// TIA Portal project "FanGas_Combustion" (V17)

(* hardware
DEVICE "PLC_1"  S7-1200 Station
   slot 0: "Rack_0"  S7-1200 Rack  Rack  V1.0
   slot 1: "PLC_1"  CPU 1214C AC/DC/Rly  6ES7 214-1BG40-0XB0  V4.5
*)

// ===== PLC "PLC_1"  CPU 1214C AC/DC/Rly =====

VAR_GLOBAL   // PLC tag table "PLC_tags"
   "风机运行" AT %Q4.4 : Bool;
   "烧嘴电源" AT %Q4.6 : Bool;
   "风机控制" AT %QW44 : Int;
END_VAR

DATA_BLOCK "信号数据"   // DB1
{ S7_Optimized_Access := 'TRUE' }
VERSION : 0.1
   VAR
      风机运行按 : Bool;   // 风机运行按钮
      风机故障反馈 : Bool;   // 风机故障反馈信号
      风机手动 : Bool;   // 风机手动模式选择
      风机自动输出 : Real;   // 风机自动控制输出值
      风机手动频率 : Real;   // 风机手动频率设定
      风机控制输出 : Real;   // 风机最终控制输出
      风压测量值 : Real;   // 风压传感器测量值
   END_VAR
BEGIN
END_DATA_BLOCK

DATA_BLOCK "内部数据"   // DB2
{ S7_Optimized_Access := 'TRUE' }
VERSION : 0.1
   VAR
      风机控制输出值 : Real;   // 风机频率百分比对应的0-27648中间值
      风压过渡 : Int;   // 风压模拟量输出过渡值
   END_VAR
BEGIN
END_DATA_BLOCK

FUNCTION "FC_FanGasControl" : Void   // FC1, LAD
{ S7_Optimized_Access := 'TRUE' }
BEGIN

REGION Network 1: 风机输出
   // 风机运行按常开+风机故障反馈常闭→风机运行线圈；手动选择MOVE自动输出或MUL手动频率×2→控制输出
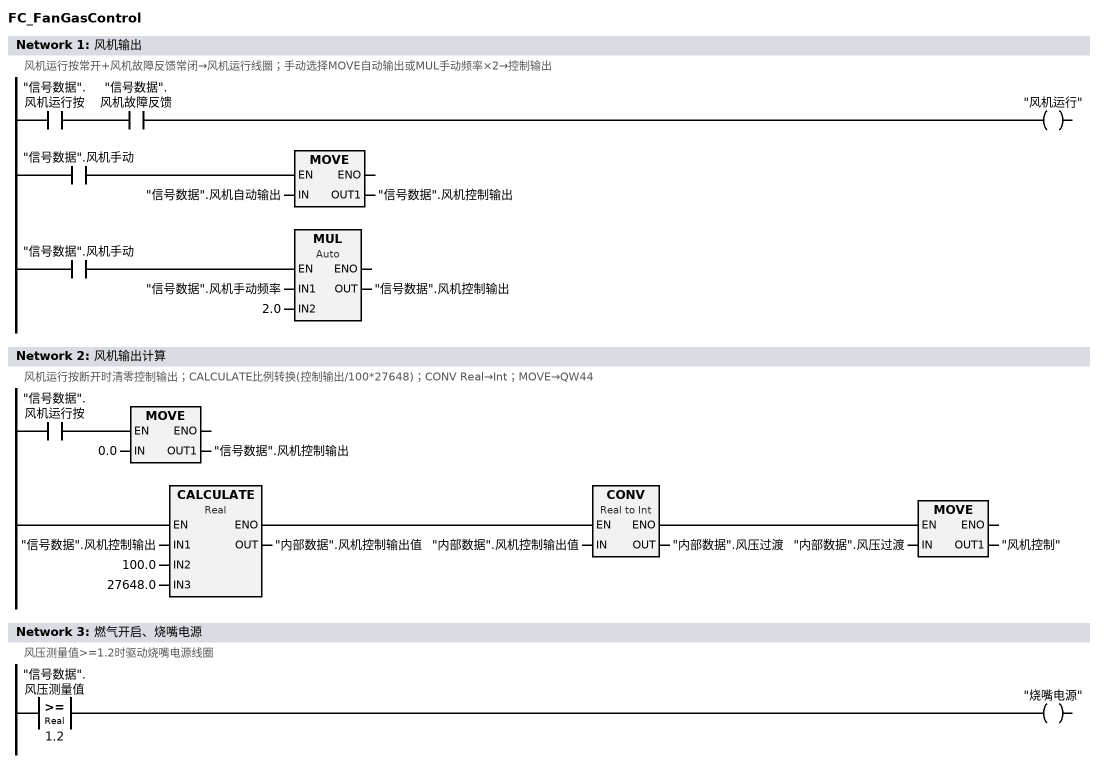
   RUNG wire#powerrail
      Contact( "信号数据".风机运行按 )
      Contact( "信号数据".风机故障反馈 )
      Coil( "风机运行" )
   END_RUNG
   RUNG wire#powerrail
      Contact( "信号数据".风机手动 )
      Move(in := "信号数据".风机自动输出, out1 => "信号数据".风机控制输出)
   END_RUNG
   RUNG wire#powerrail
      Contact( "信号数据".风机手动 )
      Mul(in1 := "信号数据".风机手动频率, in2 := 2.0, out => "信号数据".风机控制输出)
   END_RUNG
   // the same network as SCL:
   "风机运行" := "信号数据".风机运行按 AND "信号数据".风机故障反馈;
   IF "信号数据".风机手动 THEN
       "信号数据".风机控制输出 := "信号数据".风机自动输出;
       "信号数据".风机控制输出 := "信号数据".风机手动频率 * 2.0;
   END_IF;
END_REGION

REGION Network 2: 风机输出计算
   // 风机运行按断开时清零控制输出；CALCULATE比例转换(控制输出/100*27648)；CONV Real→Int；MOVE→QW44
   RUNG wire#powerrail
      Contact( "信号数据".风机运行按 )
      Move(in := 0.0, out1 => "信号数据".风机控制输出)
   END_RUNG
   RUNG wire#powerrail
      { S7_Templates := "SrcType := Real"; S7_Expression := "(IN1/IN2)*IN3" } Calculate(in1 := "信号数据".风机控制输出, in2 := 100.0, in3 := 27648.0, out => "内部数据".风机控制输出值)
      { S7_Templates := "[SrcType := Real, DestType := Int]" } Convert(in := "内部数据".风机控制输出值, out => "内部数据".风压过渡)
      Move(in := "内部数据".风压过渡, out1 => "风机控制")
   END_RUNG
   // the same network as SCL:
   IF "信号数据".风机运行按 THEN "信号数据".风机控制输出 := 0.0; END_IF;
   "内部数据".风机控制输出值 := ("信号数据".风机控制输出/100.0)*27648.0;
   "内部数据".风压过渡 := REAL_TO_INT("内部数据".风机控制输出值);
   "风机控制" := "内部数据".风压过渡;
END_REGION

REGION Network 3: 燃气开启、烧嘴电源
   // 风压测量值>=1.2时驱动烧嘴电源线圈
   RUNG wire#powerrail
      { S7_Templates := "SrcType := Real" } GE_Contact(in1 := "信号数据".风压测量值, in2 := 1.2)
      Coil( "烧嘴电源" )
   END_RUNG
   // the same network as SCL:
   "烧嘴电源" := "信号数据".风压测量值 >= 1.2;
END_REGION
END_FUNCTION

ORGANIZATION_BLOCK "Main"   // OB1, LAD, ProgramCycle
TITLE = "Main Program Sweep (Cycle)"
{ S7_Optimized_Access := 'TRUE' }
VERSION : 0.1
   VAR_INPUT
      Initial_Call : Bool;   // Initial call of this OB
      Remanence : Bool;   // =True, if remanent data are available
   END_VAR
BEGIN
END_ORGANIZATION_BLOCK